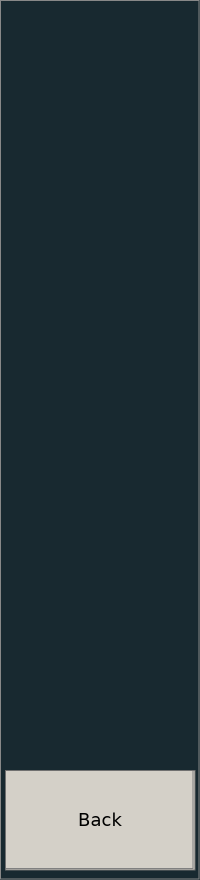
VISUALIZATION NavBarUtilities_1  // 200x880
VAR_IN_OUT
	btnBack : BOOL;
END_VAR
    Button (5,770 190x100), "Back"
        tap btnBack
END_VISUALIZATION

(* stored: Version 1.1.0.1, ProductVersion 3.1.4024.12
   Visu NavBarUtilities_1: Id {290cc033-f3ea-47d9-a038-d7754c05e74c} *)
